// Mitsubishi GX Works2 project: MAIN   PLC: FX3U/FX3UC

PROGRAM MAIN
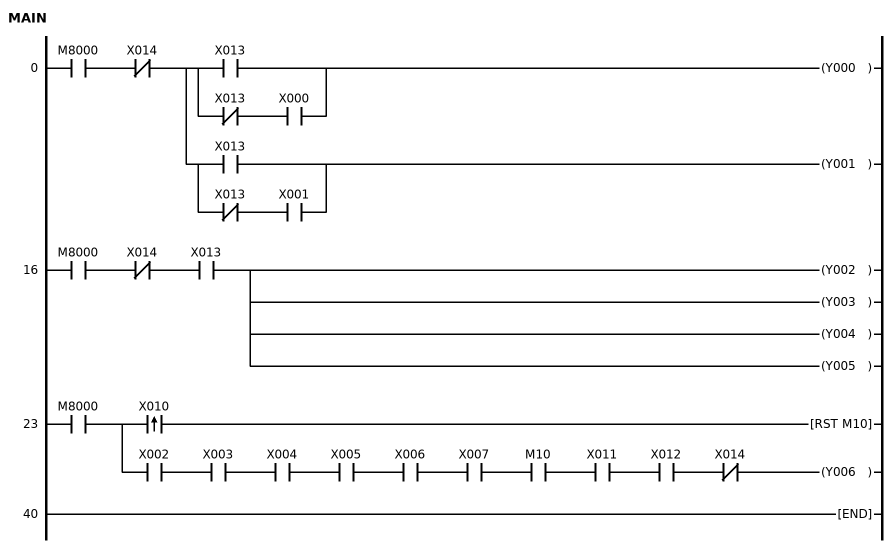
0     LD      M8000
      ANI     X014
      MPS
      LD      X013
      LDI     X013
      AND     X000
      ORB
      ANB
      OUT     Y000
      MPP
      LD      X013
      LDI     X013
      AND     X001
      ORB
      ANB
      OUT     Y001
16    LD      M8000
      ANI     X014
      AND     X013
      OUT     Y002
      OUT     Y003
      OUT     Y004
      OUT     Y005
23    LD      M8000
      MPS
      ANDP    X010
      RST     M10
      MPP
      AND     X002
      AND     X003
      AND     X004
      AND     X005
      AND     X006
      AND     X007
      AND     M10
      AND     X011
      AND     X012
      ANI     X014
      OUT     Y006
40    END
END_PROGRAM
